FUNCTION_BLOCK FT_PT2 (* 2nd grade filter with programmable times *)
  (* Standard: 61499-1 *)
  (* Version 1.5, 2025-12-21, Franz Höpfinger *)
  PACKAGE OSCAT::Basic::POUs::Engineering::Control;
  IMPORT eclipse4diac::core::TypeHash;
  IMPORT OSCAT::Basic::POUs::conversion::TIME_TO_REAL;
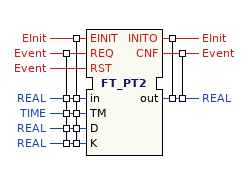
  EVENT_INPUT
    EINIT : EInit WITH in, TM, D, K; (* Init Request *)
    REQ WITH in, TM, D, K; (* Normal Execution Request *)
    RST; (* Reset Filter *)
  END_EVENT
  EVENT_OUTPUT
    INITO : EInit WITH out; (* Init Confirmation *)
    CNF WITH out; (* Execution Confirmation *)
  END_EVENT
  VAR_INPUT
    in : REAL; (* Input Signal *)
    TM : TIME; (* Time Constant *)
    D : REAL; (* Damping Factor *)
    K : REAL := 1.0; (* Gain *)
  END_VAR
  VAR_OUTPUT
    out : REAL; (* Filtered Output *)
  END_VAR
  VAR
    init : BOOL := FALSE;
    TN : REAL;
    I1 : REAL;
    I2 : REAL;
    tn2 : REAL;
  END_VAR
  FBS
    int1 : OSCAT::Basic::POUs::Engineering::Control::INTEGRATE;
    int2 : OSCAT::Basic::POUs::Engineering::Control::INTEGRATE;
  END_FBS
  EC_STATES
    EINIT : EINIT -> INITO;
    REQ : REQ -> CNF;
    RST : RST -> CNF;
  END_STATES
  ALGORITHM EINIT IN ST:
(* Startup Initialization *)
init := FALSE;
  END_ALGORITHM
  ALGORITHM RST IN ST:
init := TRUE;
out := K * in;
I2 := out;
  END_ALGORITHM
  ALGORITHM REQ IN ST:
(* startup initialisation *)
IF NOT init OR TM = T#0s THEN
	this.RST();
ELSE
	TN := TIME_TO_REAL(TM) * 1.0E-3;
	tn2 := TN * TN;
	int1.REQ(X := in * K / tn2 - I1 * 0.5 * D / TN - I2 / tn2, Y := I1);
	int2.REQ(X := I1, Y := I2);
	out := I2;
END_IF;
  END_ALGORITHM
END_FUNCTION_BLOCK
